FUNCTION_BLOCK fb_testTest EXTENDS fb_test IMPLEMENTS Testbench.IUnitTest

METHOD Test_CheckCount
VAR_INPUT
  assertions : Testbench.IAssertions;
END_VAR
VAR CONSTANT
  amsNetId : Tc2_System.T_AmsNetID := '5.5.5.5.1.1';
  deviceId : UDINT := 9;
END_VAR
Count(1);
assertions.EqualsUint(1,SUPER^.o_ui_countValue,'Value not 1');
Count(2);
assertions.EqualsUint(3,SUPER^.o_ui_countValue,'Value not 3');
END_METHOD

END_FUNCTION_BLOCK

(* stored: Version 1.1.0.1
   POU fb_testTest: Id {07648f02-c3bb-4b42-8587-c50362c01051}, SpecialFunc None
   Method Test_CheckCount: Id {4cc048b3-3e23-43a4-8a8e-3d68cc51dd91} *)
